FUNCTION_BLOCK FB_BaseStrategyController
VAR_INPUT
	stAmbientState : ST_AmbientState;
	//temperature inputs from thermal networks
	fTemperature_CN : REAL;
	fTemperature_HNLT : REAL;
	fTemperature_HNHT : REAL;
END_VAR
VAR_OUTPUT	
	//outputs for cooling network
	fTargetTemperature_CN : REAL;
	bAlgorithmPermission_CN : BOOL;
	bSetStatusOn_eChiller : BOOL;
	bLoading_CN_HVFAStorage : BOOL;
	bSetStatusOn_CN_HVFAStorage : BOOL;
	
	//outputs for low temperature heating network
	fTargetTemperature_HNLT : REAL;
	bAlgorithmPermission_HNLT : BOOL;
	bSetStatusOn_OuterCapillaryTubeMats : BOOL;
	
	//outputs for linkage systems
	bSetStatusOn_HeatPump : BOOL;
	
	//outputs for high temperature heating network
	fTargetTemperature_HNHT : REAL;
	bAlgorithmPermission_HNHT : BOOL;
	
END_VAR
VAR
	//temperature limits for thermal networks
	aTemperatureLimits_HNHT : ARRAY[1..2] OF REAL := [70,90]; //temperature limits for high temperature heating network
	aTemperatureLimits_HNLT : ARRAY[1..2] OF REAL := [30,45]; //temperature limits for low temperature heating network
	aTemperatureLimits_CN : ARRAY[1..2] OF REAL := [5,25]; //temperature limits for cooling network

	//controllers for cooling network
	Controller_eChiller : FB_CTRL_2POINT;
	Controller_eChiller_Parameters : ST_CTRL_2POINT_PARAMS;
	Controller_HVFA_CN : FB_CTRL_2POINT;
	Controller_HVFA_CN_Parameters : ST_CTRL_2POINT_PARAMS;
	bEnable_HVFA_CN : BOOL;
	
	//controllers for low temperature heating network
	Controller_OuterCapillaryTubeMats : FB_CTRL_2POINT;
	Controller_OuterCapillaryTubeMats_Parameters : ST_CTRL_2POINT_PARAMS;
	
	//controllers for hnlt and cn linkage
	Controller_HeatPump : FB_CTRL_2POINT;
	Controller_HeatPump_Parameters : ST_CTRL_2POINT_PARAMS;
END_VAR

SetTargetTemperatures();
CheckAlgorithmPermission();
ControlCN();
ControlHNLT();
ControlHnltCnLinkage();

METHOD CheckAlgorithmPermission : BOOL
VAR_INPUT
END_VAR
VAR
END_VAR
//check for algorithm permissions
bAlgorithmPermission_CN := Limiter(fInput := fTemperature_CN,fLowerLimit := aTemperatureLimits_CN[1],fUpperLimit := aTemperatureLimits_CN[2]);
bAlgorithmPermission_HNLT := Limiter(fInput := fTemperature_HNLT, fLowerLimit := aTemperatureLimits_HNLT[1], fUpperLimit := aTemperatureLimits_HNLT[2]);
bAlgorithmPermission_HNHT := Limiter(fInput := fTemperature_HNHT, fLowerLimit := aTemperatureLimits_HNHT[1], fUpperLimit := aTemperatureLimits_HNHT[2]);
END_METHOD

METHOD ControlCN : BOOL
VAR_INPUT
END_VAR
//set hysteresis parameters for two-point controllers in cooling network
Controller_eChiller_Parameters.fHysteresisRange := 4;
Controller_eChiller_Parameters.tCtrlCycleTime := GlobalVariables.tTaskCycleTime_MAIN;
Controller_eChiller_Parameters.tTaskCycleTime := GlobalVariables.tTaskCycleTime_MAIN;

//control strategy for cooling network - fSetpointValue and fActualValue are changed for cooling applications
Controller_eChiller(fSetpointValue := fTemperature_CN,
	fActualValue := fTargetTemperature_CN+2,
	eMode := eCTRL_MODE_ACTIVE,
	stParams := Controller_eChiller_Parameters);
bSetStatusOn_eChiller := Controller_eChiller.bOut;

//control hvfa storage
END_METHOD

METHOD ControlHNLT : BOOL
VAR_INPUT
END_VAR
//set hysteresis parameters for two-point controllers in cooling network
Controller_OuterCapillaryTubeMats_Parameters.fHysteresisRange := 4;
Controller_OuterCapillaryTubeMats_Parameters.tCtrlCycleTime := GlobalVariables.tTaskCycleTime_MAIN;
Controller_OuterCapillaryTubeMats_Parameters.tTaskCycleTime := GlobalVariables.tTaskCycleTime_MAIN;

//control strategy for cooling network - fSetpointValue and fActualValue are changed for cooling applications
Controller_OuterCapillaryTubeMats(fSetpointValue := fTemperature_HNLT,
	fActualValue := aTemperatureLimits_HNLT[2],
	eMode := eCTRL_MODE_ACTIVE,
	stParams := Controller_OuterCapillaryTubeMats_Parameters);
bSetStatusOn_OuterCapillaryTubeMats := Controller_OuterCapillaryTubeMats.bOut;
END_METHOD

METHOD ControlHnltCnLinkage : BOOL
VAR_INPUT
END_VAR
//set hysteresis parameters for hnlt cn linkage systems
Controller_HeatPump_Parameters.fHysteresisRange := 4;
Controller_HeatPump_Parameters.tCtrlCycleTime := GlobalVariables.tTaskCycleTime_MAIN;
Controller_HeatPump_Parameters.tTaskCycleTime := GlobalVariables.tTaskCycleTime_MAIN;

Controller_HeatPump(fSetpointValue := fTemperature_CN,
	fActualValue := fTargetTemperature_CN,
	eMode := eCTRL_MODE_ACTIVE,
	stParams := Controller_HeatPump_Parameters);
bSetStatusOn_HeatPump := Controller_HeatPump.bOut;
END_METHOD

METHOD SetTargetTemperatures : BOOL
VAR_INPUT
END_VAR
//set default target temperatures
fTargetTemperature_CN := 15;
fTargetTemperature_HNLT := 40;
fTargetTemperature_HNHT := 70;
END_METHOD

END_FUNCTION_BLOCK

(* stored: Version 1.1.0.1, ProductVersion 3.1.4024.10
   POU FB_BaseStrategyController: Id {2cc24fef-e41e-40c1-8491-4b4c0461b6c2}, SpecialFunc None
   Method CheckAlgorithmPermission: Id {66275845-0f5f-4b5e-bd16-5cacbde5e92b}
   Method ControlCN: Id {c114617d-ff2b-491a-a80e-d1c974ffb859}
   Method ControlHNLT: Id {57bcb54f-1f56-4d59-8bc6-dbfcc2a5773d}
   Method ControlHnltCnLinkage: Id {47fe50a8-fa6a-42c9-86f6-4129fa6636fe}
   Method SetTargetTemperatures: Id {6be7450f-8e0b-4497-9741-f2ddcfb682eb} *)
